SUBAPPLICATION Uebung_006a2_AX (* 2x SR und T-Flip-Flop mit IE *)
  (* Standard: 61499-2; Description: Copyright (c) 2023 Meisterschulen am Ostbahnhof This program and the accompanying materials are made available under the terms of the Eclipse Public License 2.0 which is available at https://www.eclipse.org/legal/epl-2.0/ SPDX-License-Identifier: EPL-2.0 *)
  (* Version 1.0, 2026-01-13, Franz Höpfinger, Meisterschulen am Ostbahnhof, initial API and implementation and/or initial documentation *)
  PACKAGE Uebungen;
  IMPORT logiBUS::io::DI::logiBUS_DI::Input_I1;
  IMPORT logiBUS::io::DI::logiBUS_DI::Input_I2;
  IMPORT logiBUS::io::DI::logiBUS_DI::Input_I3;
  IMPORT logiBUS::io::DI::logiBUS_DI_Events::BUTTON_SINGLE_CLICK;
  IMPORT logiBUS::io::DQ::logiBUS_DO::Output_Q1;
  IMPORT logiBUS::io::DQ::logiBUS_DO::Output_Q2;
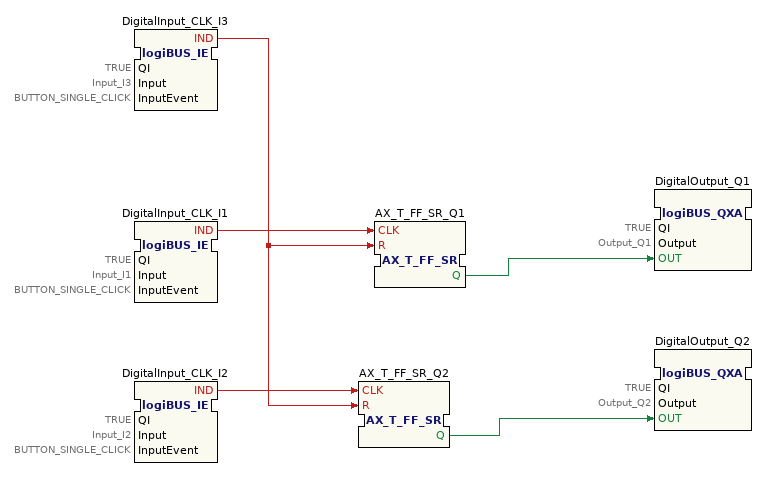
  FBS
    DigitalOutput_Q1 : logiBUS::io::DQ::logiBUS_QXA(QI := TRUE, Output := Output_Q1);
    DigitalInput_CLK_I1 : logiBUS::io::DI::logiBUS_IE(QI := TRUE, Input := Input_I1, InputEvent := BUTTON_SINGLE_CLICK);
    DigitalInput_CLK_I2 : logiBUS::io::DI::logiBUS_IE(QI := TRUE, Input := Input_I2, InputEvent := BUTTON_SINGLE_CLICK);
    AX_T_FF_SR_Q1 : adapter::events::unidirectional::AX_T_FF_SR;
    DigitalInput_CLK_I3 : logiBUS::io::DI::logiBUS_IE(QI := TRUE, Input := Input_I3, InputEvent := BUTTON_SINGLE_CLICK);
    AX_T_FF_SR_Q2 : adapter::events::unidirectional::AX_T_FF_SR;
    DigitalOutput_Q2 : logiBUS::io::DQ::logiBUS_QXA(QI := TRUE, Output := Output_Q2);
  END_FBS
  EVENT_CONNECTIONS
    DigitalInput_CLK_I1.IND TO AX_T_FF_SR_Q1.CLK;
    DigitalInput_CLK_I2.IND TO AX_T_FF_SR_Q2.CLK;
    DigitalInput_CLK_I3.IND TO AX_T_FF_SR_Q2.R;
    DigitalInput_CLK_I3.IND TO AX_T_FF_SR_Q1.R;
  END_CONNECTIONS
  ADAPTER_CONNECTIONS
    AX_T_FF_SR_Q1.Q TO DigitalOutput_Q1.OUT;
    AX_T_FF_SR_Q2.Q TO DigitalOutput_Q2.OUT;
  END_CONNECTIONS
END_SUBAPPLICATION
